// TwinCAT 3 PLC project curve_editor_PLC
// ProgramVersion: 3.1.4026.17
// libraries:
//   Tc2_Standard, * (Beckhoff Automation GmbH)
//   Tc2_System, * (Beckhoff Automation GmbH)
// project tree:
//   DUTs/ CPoint.TcDUT (not stored)
//   GVLs/ GVL.TcGVL (not stored)
//   / PlcTask.TcTTO
//   POUs/CurveEditor/ FB_CamWTC.TcPOU (not stored)
//   POUs/ MAIN.TcPOU

CONFIGURATION curve_editor_PLC
    RESOURCE PLC ON TwinCAT3
        TASK PlcTask(INTERVAL := T#10ms, PRIORITY := 20);
        PROGRAM MAIN WITH PlcTask : MAIN;
    END_RESOURCE
END_CONFIGURATION

// ---- POUs/MAIN.TcPOU
PROGRAM MAIN
VAR
						
	// CurveEditor Varaibles
	fbWTC1: FB_CamWTC;
	fbWTC2: FB_CamWTC;
END_VAR

fbWTC1();
fbWTC2();

END_PROGRAM
